// TIA Portal V20 export
// export: Created 2026-07-10T11:12:27.8616587Z, ExportSetting WithDefaults, DisplayName Totally Integrated Automation Portal, DisplayVersion V20, DisplayName TIA Portal Openness, DisplayVersion V20, DisplayName TIA Portal Version Control Interface, DisplayVersion V20, DisplayName STEP 7 Professional, DisplayVersion V20, DisplayName STEP 7 Safety, DisplayVersion V20, DisplayName WinCC Basic/Comfort/Advanced, DisplayVersion V20, DisplayName WinCC Unified, DisplayVersion V20
DATA_BLOCK "Alarms_DB"   // DB11
VERSION : 0.1
// stored: AutoNumber true, DBAccessibleFromOPCUA true, InstanceOfName Alarms, InstanceOfType FB
"Alarms"
   // VAR
   //    WaterOutMaxTON { S7_SetPoint := 'True'} : TON_TIME;
   //    WaterOutMinTON { S7_SetPoint := 'True'} : TON_TIME;
   //    WaterInMaxTON { S7_SetPoint := 'True'} : TON_TIME;
   //    WaterInMinTON { S7_SetPoint := 'True'} : TON_TIME;
   //    "step" { S7_SetPoint := 'True'} : Int;
   //    ChlorAlarm { S7_SetPoint := 'True'} : "ChlorConsumptionAlarm";
   // END_VAR
BEGIN
   WaterOutMaxTON.PT := T#0MS;
   WaterOutMaxTON.IN := TRUE;
   WaterOutMinTON.PT := T#0MS;
   WaterOutMinTON.IN := TRUE;
END_DATA_BLOCK
